FUNCTION_BLOCK PWMChip (* Configures one Linux PWM channel (/sys/class/pwm) as the IO handle VALUE for a QW *)
  (* Description: Copyright (c) 2026 Aalborg University This program and the accompanying materials are made available under the terms of the Eclipse Public License 2.0 which is available at https://www.eclipse.org/legal/epl-2.0/ SPDX-License-Identifier: EPL-2.0 *)
  (* Version 1.0, 2026-09-29, Martin Jensen, Aalborg University, FORTE module pwmsysfs (4diac/tools/forte-patches) *)
  PACKAGE eclipse4diac::io::pwmsysfs;
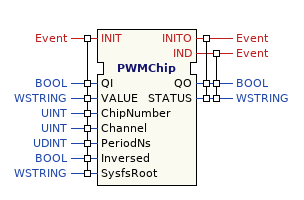
  EVENT_INPUT
    INIT WITH QI, VALUE, ChipNumber, Channel, PeriodNs, Inversed, SysfsRoot; (* Service Initialization *)
  END_EVENT
  EVENT_OUTPUT
    INITO WITH QO, STATUS; (* Initialization Confirm *)
    IND WITH QO, STATUS; (* Indication from Resource *)
  END_EVENT
  VAR_INPUT
    QI : BOOL; (* Event Input Qualifier *)
    VALUE : WSTRING; (* Handle name the QW refers to (its PARAMS) *)
    ChipNumber : UINT := 0; (* N of /sys/class/pwm/pwmchipN *)
    Channel : UINT := 0; (* Channel of the chip (pwmM) *)
    PeriodNs : UDINT := 1000000; (* Period in ns (1000000 = 1 kHz, 20000000 = 50 Hz for servos) *)
    Inversed : BOOL := FALSE; (* Inversed polarity *)
    SysfsRoot : WSTRING; (* Default /sys/class/pwm (another folder for tests) *)
  END_VAR
  VAR_OUTPUT
    QO : BOOL; (* Event Output Qualifier *)
    STATUS : WSTRING; (* Service Status *)
  END_VAR
END_FUNCTION_BLOCK
